//
point										:= 42;
_Camming.camPoints[point].MasterPos			:= 1030.100;
_Camming.camPoints[point].SlavePos			:= 916.716;
_Camming.camPoints[point].PointIndex		:= point;
_Camming.camPoints[point].FunctionType		:= MC_MotionFunctionType.MOTIONFUNCTYPE_POLYNOM5_MM;
_Camming.camPoints[point].PointType			:= MC_MotionPointType.MOTIONPOINTTYPE_MOTION;
_Camming.camPoints[point].RelIndexNextPoint := 1;
_Camming.camPoints[point].SlaveVelo			:= 1.187356;
_Camming.camPoints[point].SlaveAcc			:= 0.01442322;
_Camming.camPoints[point].SlaveJerk			:= 0.00;

//
point										:= 43;
_Camming.camPoints[point].MasterPos			:= 1039.967;
_Camming.camPoints[point].SlavePos			:= 929.194;
_Camming.camPoints[point].PointIndex		:= point;
_Camming.camPoints[point].FunctionType		:= MC_MotionFunctionType.MOTIONFUNCTYPE_POLYNOM5_MM;
_Camming.camPoints[point].PointType			:= MC_MotionPointType.MOTIONPOINTTYPE_MOTION;
_Camming.camPoints[point].RelIndexNextPoint := 1;
_Camming.camPoints[point].SlaveVelo			:= 1.346759;
_Camming.camPoints[point].SlaveAcc			:= 0.01732695;
_Camming.camPoints[point].SlaveJerk			:= 0.00;

//
point										:= 44;
_Camming.camPoints[point].MasterPos			:= 1049.833;
_Camming.camPoints[point].SlavePos			:= 943.327;
_Camming.camPoints[point].PointIndex		:= point;
_Camming.camPoints[point].FunctionType		:= MC_MotionFunctionType.MOTIONFUNCTYPE_POLYNOM5_MM;
_Camming.camPoints[point].PointType			:= MC_MotionPointType.MOTIONPOINTTYPE_MOTION;
_Camming.camPoints[point].RelIndexNextPoint := 1;
_Camming.camPoints[point].SlaveVelo			:= 1.516335;
_Camming.camPoints[point].SlaveAcc			:= 0.01633779;
_Camming.camPoints[point].SlaveJerk			:= 0.00;

//
point										:= 45;
_Camming.camPoints[point].MasterPos			:= 1059.700;
_Camming.camPoints[point].SlavePos			:= 959.017;
_Camming.camPoints[point].PointIndex		:= point;
_Camming.camPoints[point].FunctionType		:= MC_MotionFunctionType.MOTIONFUNCTYPE_POLYNOM5_MM;
_Camming.camPoints[point].PointType			:= MC_MotionPointType.MOTIONPOINTTYPE_MOTION;
_Camming.camPoints[point].RelIndexNextPoint := 1;
_Camming.camPoints[point].SlaveVelo			:= 1.655944;
_Camming.camPoints[point].SlaveAcc			:= 0.01140889;
_Camming.camPoints[point].SlaveJerk			:= 0.00;

//
point										:= 46;
_Camming.camPoints[point].MasterPos			:= 1069.567;
_Camming.camPoints[point].SlavePos			:= 975.802;
_Camming.camPoints[point].PointIndex		:= point;
_Camming.camPoints[point].FunctionType		:= MC_MotionFunctionType.MOTIONFUNCTYPE_POLYNOM5_MM;
_Camming.camPoints[point].PointType			:= MC_MotionPointType.MOTIONPOINTTYPE_MOTION;
_Camming.camPoints[point].RelIndexNextPoint := 1;
_Camming.camPoints[point].SlaveVelo			:= 1.735262;
_Camming.camPoints[point].SlaveAcc			:= 0.00466021;
_Camming.camPoints[point].SlaveJerk			:= 0.00;

//
point										:= 47;
_Camming.camPoints[point].MasterPos			:= 1079.433;
_Camming.camPoints[point].SlavePos			:= 993.059;
_Camming.camPoints[point].PointIndex		:= point;
_Camming.camPoints[point].FunctionType		:= MC_MotionFunctionType.MOTIONFUNCTYPE_POLYNOM5_MM;
_Camming.camPoints[point].PointType			:= MC_MotionPointType.MOTIONPOINTTYPE_MOTION;
_Camming.camPoints[point].RelIndexNextPoint := 1;
_Camming.camPoints[point].SlaveVelo			:= 1.755026;
_Camming.camPoints[point].SlaveAcc			:= 0.00009489;
_Camming.camPoints[point].SlaveJerk			:= 0.00;

//
point										:= 48;
_Camming.camPoints[point].MasterPos			:= 1089.300;
_Camming.camPoints[point].SlavePos			:= 1010.346;
_Camming.camPoints[point].PointIndex		:= point;
_Camming.camPoints[point].FunctionType		:= MC_MotionFunctionType.MOTIONFUNCTYPE_POLYNOM5_MM;
_Camming.camPoints[point].PointType			:= MC_MotionPointType.MOTIONPOINTTYPE_MOTION;
_Camming.camPoints[point].RelIndexNextPoint := 1;
_Camming.camPoints[point].SlaveVelo			:= 1.737154;
_Camming.camPoints[point].SlaveAcc			:= -0.00845956;
_Camming.camPoints[point].SlaveJerk			:= 0.00;

//
point										:= 49;
_Camming.camPoints[point].MasterPos			:= 1099.167;
_Camming.camPoints[point].SlavePos			:= 1026.699;
_Camming.camPoints[point].PointIndex		:= point;
_Camming.camPoints[point].FunctionType		:= MC_MotionFunctionType.MOTIONFUNCTYPE_POLYNOM5_MM;
_Camming.camPoints[point].PointType			:= MC_MotionPointType.MOTIONPOINTTYPE_MOTION;
_Camming.camPoints[point].RelIndexNextPoint := 1;
_Camming.camPoints[point].SlaveVelo			:= 1.547397;
_Camming.camPoints[point].SlaveAcc			:= -0.02615257;
_Camming.camPoints[point].SlaveJerk			:= 0.00;

//
point										:= 50;
_Camming.camPoints[point].MasterPos			:= 1109.033;
_Camming.camPoints[point].SlavePos			:= 1040.717;
_Camming.camPoints[point].PointIndex		:= point;
_Camming.camPoints[point].FunctionType		:= MC_MotionFunctionType.MOTIONFUNCTYPE_POLYNOM5_MM;
_Camming.camPoints[point].PointType			:= MC_MotionPointType.MOTIONPOINTTYPE_MOTION;
_Camming.camPoints[point].RelIndexNextPoint := 1;
_Camming.camPoints[point].SlaveVelo			:= 1.302751;
_Camming.camPoints[point].SlaveAcc			:= -0.02131854;
_Camming.camPoints[point].SlaveJerk			:= 0.00;

//
point										:= 51;
_Camming.camPoints[point].MasterPos			:= 1118.900;
_Camming.camPoints[point].SlavePos			:= 1052.681;
_Camming.camPoints[point].PointIndex		:= point;
_Camming.camPoints[point].FunctionType		:= MC_MotionFunctionType.MOTIONFUNCTYPE_POLYNOM5_MM;
_Camming.camPoints[point].PointType			:= MC_MotionPointType.MOTIONPOINTTYPE_MOTION;
_Camming.camPoints[point].RelIndexNextPoint := 1;
_Camming.camPoints[point].SlaveVelo			:= 1.136789;
_Camming.camPoints[point].SlaveAcc			:= -0.01261846;
_Camming.camPoints[point].SlaveJerk			:= 0.00;

//
point										:= 52;
_Camming.camPoints[point].MasterPos			:= 1128.767;
_Camming.camPoints[point].SlavePos			:= 1063.397;
_Camming.camPoints[point].PointIndex		:= point;
_Camming.camPoints[point].FunctionType		:= MC_MotionFunctionType.MOTIONFUNCTYPE_POLYNOM5_MM;
_Camming.camPoints[point].PointType			:= MC_MotionPointType.MOTIONPOINTTYPE_MOTION;
_Camming.camPoints[point].RelIndexNextPoint := 1;
_Camming.camPoints[point].SlaveVelo			:= 1.045962;
_Camming.camPoints[point].SlaveAcc			:= -0.00622413;
_Camming.camPoints[point].SlaveJerk			:= 0.00;

//
point										:= 53;
_Camming.camPoints[point].MasterPos			:= 1138.633;
_Camming.camPoints[point].SlavePos			:= 1073.492;
_Camming.camPoints[point].PointIndex		:= point;
_Camming.camPoints[point].FunctionType		:= MC_MotionFunctionType.MOTIONFUNCTYPE_POLYNOM5_MM;
_Camming.camPoints[point].PointType			:= MC_MotionPointType.MOTIONPOINTTYPE_MOTION;
_Camming.camPoints[point].RelIndexNextPoint := 1;
_Camming.camPoints[point].SlaveVelo			:= 1.007263;
_Camming.camPoints[point].SlaveAcc			:= -0.00195545;
_Camming.camPoints[point].SlaveJerk			:= 0.00;

//
point										:= 54;
_Camming.camPoints[point].MasterPos			:= 1148.500;
_Camming.camPoints[point].SlavePos			:= 1083.378;
_Camming.camPoints[point].PointIndex		:= point;
_Camming.camPoints[point].FunctionType		:= MC_MotionFunctionType.MOTIONFUNCTYPE_POLYNOM5_MM;
_Camming.camPoints[point].PointType			:= MC_MotionPointType.MOTIONPOINTTYPE_MOTION;
_Camming.camPoints[point].RelIndexNextPoint := 1;
_Camming.camPoints[point].SlaveVelo			:= 1.000000;
_Camming.camPoints[point].SlaveAcc			:= 0.00000000;
_Camming.camPoints[point].SlaveJerk			:= 0.00;

//
point										:= 55;
_Camming.camPoints[point].MasterPos			:= 1416.600;
_Camming.camPoints[point].SlavePos			:= 1351.478;
_Camming.camPoints[point].PointIndex		:= point;
_Camming.camPoints[point].FunctionType		:= MC_MotionFunctionType.MOTIONFUNCTYPE_POLYNOM5_MM;
_Camming.camPoints[point].PointType			:= MC_MotionPointType.MOTIONPOINTTYPE_MOTION;
_Camming.camPoints[point].RelIndexNextPoint := 1;
_Camming.camPoints[point].SlaveVelo			:= 1.000000;
_Camming.camPoints[point].SlaveAcc			:= 0.00000000;
_Camming.camPoints[point].SlaveJerk			:= 0.00;

//
point										:= 56;
_Camming.camPoints[point].MasterPos			:= 1426.495;
_Camming.camPoints[point].SlavePos			:= 1361.354;
_Camming.camPoints[point].PointIndex		:= point;
_Camming.camPoints[point].FunctionType		:= MC_MotionFunctionType.MOTIONFUNCTYPE_POLYNOM5_MM;
_Camming.camPoints[point].PointType			:= MC_MotionPointType.MOTIONPOINTTYPE_MOTION;
_Camming.camPoints[point].RelIndexNextPoint := 1;
_Camming.camPoints[point].SlaveVelo			:= 0.992814;
_Camming.camPoints[point].SlaveAcc			:= -0.00190944;
_Camming.camPoints[point].SlaveJerk			:= 0.00;

//
point										:= 57;
_Camming.camPoints[point].MasterPos			:= 1436.390;
_Camming.camPoints[point].SlavePos			:= 1371.030;
_Camming.camPoints[point].PointIndex		:= point;
_Camming.camPoints[point].FunctionType		:= MC_MotionFunctionType.MOTIONFUNCTYPE_POLYNOM5_MM;
_Camming.camPoints[point].PointType			:= MC_MotionPointType.MOTIONPOINTTYPE_MOTION;
_Camming.camPoints[point].RelIndexNextPoint := 1;
_Camming.camPoints[point].SlaveVelo			:= 0.957206;
_Camming.camPoints[point].SlaveAcc			:= -0.00535633;
_Camming.camPoints[point].SlaveJerk			:= 0.00;

//
point										:= 58;
_Camming.camPoints[point].MasterPos			:= 1446.285;
_Camming.camPoints[point].SlavePos			:= 1380.186;
_Camming.camPoints[point].PointIndex		:= point;
_Camming.camPoints[point].FunctionType		:= MC_MotionFunctionType.MOTIONFUNCTYPE_POLYNOM5_MM;
_Camming.camPoints[point].PointType			:= MC_MotionPointType.MOTIONPOINTTYPE_MOTION;
_Camming.camPoints[point].RelIndexNextPoint := 1;
_Camming.camPoints[point].SlaveVelo			:= 0.888425;
_Camming.camPoints[point].SlaveAcc			:= -0.00834680;
_Camming.camPoints[point].SlaveJerk			:= 0.00;

//
point										:= 59;
_Camming.camPoints[point].MasterPos			:= 1456.180;
_Camming.camPoints[point].SlavePos			:= 1388.538;
_Camming.camPoints[point].PointIndex		:= point;
_Camming.camPoints[point].FunctionType		:= MC_MotionFunctionType.MOTIONFUNCTYPE_POLYNOM5_MM;
_Camming.camPoints[point].PointType			:= MC_MotionPointType.MOTIONPOINTTYPE_MOTION;
_Camming.camPoints[point].RelIndexNextPoint := 1;
_Camming.camPoints[point].SlaveVelo			:= 0.797621;
_Camming.camPoints[point].SlaveAcc			:= -0.00966634;
_Camming.camPoints[point].SlaveJerk			:= 0.00;

//
point										:= 60;
_Camming.camPoints[point].MasterPos			:= 1466.075;
_Camming.camPoints[point].SlavePos			:= 1395.962;
_Camming.camPoints[point].PointIndex		:= point;
_Camming.camPoints[point].FunctionType		:= MC_MotionFunctionType.MOTIONFUNCTYPE_POLYNOM5_MM;
_Camming.camPoints[point].PointType			:= MC_MotionPointType.MOTIONPOINTTYPE_MOTION;
_Camming.camPoints[point].RelIndexNextPoint := 1;
_Camming.camPoints[point].SlaveVelo			:= 0.704244;
_Camming.camPoints[point].SlaveAcc			:= -0.00885381;
_Camming.camPoints[point].SlaveJerk			:= 0.00;

//
point										:= 61;
_Camming.camPoints[point].MasterPos			:= 1475.970;
_Camming.camPoints[point].SlavePos			:= 1402.534;
_Camming.camPoints[point].PointIndex		:= point;
_Camming.camPoints[point].FunctionType		:= MC_MotionFunctionType.MOTIONFUNCTYPE_POLYNOM5_MM;
_Camming.camPoints[point].PointType			:= MC_MotionPointType.MOTIONPOINTTYPE_MOTION;
_Camming.camPoints[point].RelIndexNextPoint := 1;
_Camming.camPoints[point].SlaveVelo			:= 0.628520;
_Camming.camPoints[point].SlaveAcc			:= -0.00621225;
_Camming.camPoints[point].SlaveJerk			:= 0.00;

//
point										:= 62;
_Camming.camPoints[point].MasterPos			:= 1485.865;
_Camming.camPoints[point].SlavePos			:= 1408.505;
_Camming.camPoints[point].PointIndex		:= point;
_Camming.camPoints[point].FunctionType		:= MC_MotionFunctionType.MOTIONFUNCTYPE_POLYNOM5_MM;
_Camming.camPoints[point].PointType			:= MC_MotionPointType.MOTIONPOINTTYPE_MOTION;
_Camming.camPoints[point].RelIndexNextPoint := 1;
_Camming.camPoints[point].SlaveVelo			:= 0.583944;
_Camming.camPoints[point].SlaveAcc			:= -0.00279152;
_Camming.camPoints[point].SlaveJerk			:= 0.00;

//
point										:= 63;
_Camming.camPoints[point].MasterPos			:= 1495.760;
_Camming.camPoints[point].SlavePos			:= 1414.195;
_Camming.camPoints[point].PointIndex		:= point;
_Camming.camPoints[point].FunctionType		:= MC_MotionFunctionType.MOTIONFUNCTYPE_POLYNOM5_MM;
_Camming.camPoints[point].PointType			:= MC_MotionPointType.MOTIONPOINTTYPE_MOTION;
_Camming.camPoints[point].RelIndexNextPoint := 1;
_Camming.camPoints[point].SlaveVelo			:= 0.570311;
_Camming.camPoints[point].SlaveAcc			:= -0.00028497;
_Camming.camPoints[point].SlaveJerk			:= 0.00;

//
point										:= 64;
_Camming.camPoints[point].MasterPos			:= 1505.655;
_Camming.camPoints[point].SlavePos			:= 1419.834;
_Camming.camPoints[point].PointIndex		:= point;
_Camming.camPoints[point].FunctionType		:= MC_MotionFunctionType.MOTIONFUNCTYPE_POLYNOM5_MM;
_Camming.camPoints[point].PointType			:= MC_MotionPointType.MOTIONPOINTTYPE_MOTION;
_Camming.camPoints[point].RelIndexNextPoint := 1;
_Camming.camPoints[point].SlaveVelo			:= 0.569785;
_Camming.camPoints[point].SlaveAcc			:= -0.00000641;
_Camming.camPoints[point].SlaveJerk			:= 0.00;

//
point										:= 65;
_Camming.camPoints[point].MasterPos			:= 1515.550;
_Camming.camPoints[point].SlavePos			:= 1425.476;
_Camming.camPoints[point].PointIndex		:= point;
_Camming.camPoints[point].FunctionType		:= MC_MotionFunctionType.MOTIONFUNCTYPE_POLYNOM5_MM;
_Camming.camPoints[point].PointType			:= MC_MotionPointType.MOTIONPOINTTYPE_MOTION;
_Camming.camPoints[point].RelIndexNextPoint := 1;
_Camming.camPoints[point].SlaveVelo			:= 0.571122;
_Camming.camPoints[point].SlaveAcc			:= 0.00033576;
_Camming.camPoints[point].SlaveJerk			:= 0.00;

//
point										:= 66;
_Camming.camPoints[point].MasterPos			:= 1525.445;
_Camming.camPoints[point].SlavePos			:= 1431.153;
_Camming.camPoints[point].PointIndex		:= point;
_Camming.camPoints[point].FunctionType		:= MC_MotionFunctionType.MOTIONFUNCTYPE_POLYNOM5_MM;
_Camming.camPoints[point].PointType			:= MC_MotionPointType.MOTIONPOINTTYPE_MOTION;
_Camming.camPoints[point].RelIndexNextPoint := 1;
_Camming.camPoints[point].SlaveVelo			:= 0.577454;
_Camming.camPoints[point].SlaveAcc			:= 0.00098723;
_Camming.camPoints[point].SlaveJerk			:= 0.00;

//
point										:= 67;
_Camming.camPoints[point].MasterPos			:= 1535.340;
_Camming.camPoints[point].SlavePos			:= 1436.929;
_Camming.camPoints[point].PointIndex		:= point;
_Camming.camPoints[point].FunctionType		:= MC_MotionFunctionType.MOTIONFUNCTYPE_POLYNOM5_MM;
_Camming.camPoints[point].PointType			:= MC_MotionPointType.MOTIONPOINTTYPE_MOTION;
_Camming.camPoints[point].RelIndexNextPoint := 1;
_Camming.camPoints[point].SlaveVelo			:= 0.591500;
_Camming.camPoints[point].SlaveAcc			:= 0.00188997;
_Camming.camPoints[point].SlaveJerk			:= 0.00;

//
point										:= 68;
_Camming.camPoints[point].MasterPos			:= 1545.235;
_Camming.camPoints[point].SlavePos			:= 1442.892;
_Camming.camPoints[point].PointIndex		:= point;
_Camming.camPoints[point].FunctionType		:= MC_MotionFunctionType.MOTIONFUNCTYPE_POLYNOM5_MM;
_Camming.camPoints[point].PointType			:= MC_MotionPointType.MOTIONPOINTTYPE_MOTION;
_Camming.camPoints[point].RelIndexNextPoint := 1;
_Camming.camPoints[point].SlaveVelo			:= 0.615664;
_Camming.camPoints[point].SlaveAcc			:= 0.00303751;
_Camming.camPoints[point].SlaveJerk			:= 0.00;

//
point										:= 69;
_Camming.camPoints[point].MasterPos			:= 1555.130;
_Camming.camPoints[point].SlavePos			:= 1449.155;
_Camming.camPoints[point].PointIndex		:= point;
_Camming.camPoints[point].FunctionType		:= MC_MotionFunctionType.MOTIONFUNCTYPE_POLYNOM5_MM;
_Camming.camPoints[point].PointType			:= MC_MotionPointType.MOTIONPOINTTYPE_MOTION;
_Camming.camPoints[point].RelIndexNextPoint := 1;
_Camming.camPoints[point].SlaveVelo			:= 0.652442;
_Camming.camPoints[point].SlaveAcc			:= 0.00443439;
_Camming.camPoints[point].SlaveJerk			:= 0.00;

//
point										:= 70;
_Camming.camPoints[point].MasterPos			:= 1565.025;
_Camming.camPoints[point].SlavePos			:= 1455.854;
_Camming.camPoints[point].PointIndex		:= point;
_Camming.camPoints[point].FunctionType		:= MC_MotionFunctionType.MOTIONFUNCTYPE_POLYNOM5_MM;
_Camming.camPoints[point].PointType			:= MC_MotionPointType.MOTIONPOINTTYPE_MOTION;
_Camming.camPoints[point].RelIndexNextPoint := 1;
_Camming.camPoints[point].SlaveVelo			:= 0.704402;
_Camming.camPoints[point].SlaveAcc			:= 0.00609093;
_Camming.camPoints[point].SlaveJerk			:= 0.00;

//
point										:= 71;
_Camming.camPoints[point].MasterPos			:= 1574.920;
_Camming.camPoints[point].SlavePos			:= 1463.150;
_Camming.camPoints[point].PointIndex		:= point;
_Camming.camPoints[point].FunctionType		:= MC_MotionFunctionType.MOTIONFUNCTYPE_POLYNOM5_MM;
_Camming.camPoints[point].PointType			:= MC_MotionPointType.MOTIONPOINTTYPE_MOTION;
_Camming.camPoints[point].RelIndexNextPoint := 1;
_Camming.camPoints[point].SlaveVelo			:= 0.773096;
_Camming.camPoints[point].SlaveAcc			:= 0.00774577;
_Camming.camPoints[point].SlaveJerk			:= 0.00;

//
point										:= 72;
_Camming.camPoints[point].MasterPos			:= 1584.815;
_Camming.camPoints[point].SlavePos			:= 1471.200;
_Camming.camPoints[point].PointIndex		:= point;
_Camming.camPoints[point].FunctionType		:= MC_MotionFunctionType.MOTIONFUNCTYPE_POLYNOM5_MM;
_Camming.camPoints[point].PointType			:= MC_MotionPointType.MOTIONPOINTTYPE_MOTION;
_Camming.camPoints[point].RelIndexNextPoint := 1;
_Camming.camPoints[point].SlaveVelo			:= 0.855433;
_Camming.camPoints[point].SlaveAcc			:= 0.00865192;
_Camming.camPoints[point].SlaveJerk			:= 0.00;

//
point										:= 73;
_Camming.camPoints[point].MasterPos			:= 1594.710;
_Camming.camPoints[point].SlavePos			:= 1480.077;
_Camming.camPoints[point].PointIndex		:= point;
_Camming.camPoints[point].FunctionType		:= MC_MotionFunctionType.MOTIONFUNCTYPE_POLYNOM5_MM;
_Camming.camPoints[point].PointType			:= MC_MotionPointType.MOTIONPOINTTYPE_MOTION;
_Camming.camPoints[point].RelIndexNextPoint := 1;
_Camming.camPoints[point].SlaveVelo			:= 0.936508;
_Camming.camPoints[point].SlaveAcc			:= 0.00721864;
_Camming.camPoints[point].SlaveJerk			:= 0.00;

//
point										:= 74;
_Camming.camPoints[point].MasterPos			:= 1604.605;
_Camming.camPoints[point].SlavePos			:= 1489.636;
_Camming.camPoints[point].PointIndex		:= point;
_Camming.camPoints[point].FunctionType		:= MC_MotionFunctionType.MOTIONFUNCTYPE_POLYNOM5_MM;
_Camming.camPoints[point].PointType			:= MC_MotionPointType.MOTIONPOINTTYPE_MOTION;
_Camming.camPoints[point].RelIndexNextPoint := 1;
_Camming.camPoints[point].SlaveVelo			:= 0.988558;
_Camming.camPoints[point].SlaveAcc			:= 0.00301892;
_Camming.camPoints[point].SlaveJerk			:= 0.00;

//
point										:= 75;
_Camming.camPoints[point].MasterPos			:= 1614.500;
_Camming.camPoints[point].SlavePos			:= 1499.500;
_Camming.camPoints[point].PointIndex		:= point;
_Camming.camPoints[point].FunctionType		:= MC_MotionFunctionType.MOTIONFUNCTYPE_POLYNOM5_MM;
_Camming.camPoints[point].PointType			:= MC_MotionPointType.MOTIONPOINTTYPE_MOTION;
_Camming.camPoints[point].RelIndexNextPoint := 1;
_Camming.camPoints[point].SlaveVelo			:= 1.000000;
_Camming.camPoints[point].SlaveAcc			:= 0.00000000;
_Camming.camPoints[point].SlaveJerk			:= 0.00;

//
point										:= 76;
_Camming.camPoints[point].MasterPos			:= 1680.000;
_Camming.camPoints[point].SlavePos			:= 1565.000;
_Camming.camPoints[point].PointIndex		:= point;
_Camming.camPoints[point].FunctionType		:= MC_MotionFunctionType.MOTIONFUNCTYPE_POLYNOM5_MM;
_Camming.camPoints[point].PointType			:= MC_MotionPointType.MOTIONPOINTTYPE_MOTION;
_Camming.camPoints[point].RelIndexNextPoint := 0;
_Camming.camPoints[point].SlaveVelo			:= 1.000000;
_Camming.camPoints[point].SlaveAcc			:= 0.00000000;
_Camming.camPoints[point].SlaveJerk			:= 0.00;
END_METHOD

METHOD Old
VAR_INPUT
END_VAR
IF NOT _Custom THEN
	point										:= 1;
	_Camming.camPoints[point].MasterPos			:= 250;
	_Camming.camPoints[point].SlavePos			:= 135;
	_Camming.camPoints[point].PointIndex		:= point;
	_Camming.camPoints[point].FunctionType		:= MC_MotionFunctionType.MOTIONFUNCTYPE_POLYNOM1;
	_Camming.camPoints[point].PointType			:= MC_MotionPointType.MOTIONPOINTTYPE_ACTIVATION;
	_Camming.camPoints[point].RelIndexNextPoint := 1;
	_Camming.camPoints[point].SlaveVelo			:= 0.00;
	_Camming.camPoints[point].SlaveAcc			:= 0.00;
	_Camming.camPoints[point].SlaveJerk			:= 0.00;

	//
	point										:= 2;
	_Camming.camPoints[point].MasterPos			:= 291;
	_Camming.camPoints[point].SlavePos			:= 176;
	_Camming.camPoints[point].PointIndex		:= point;
	_Camming.camPoints[point].FunctionType		:= MC_MotionFunctionType.MOTIONFUNCTYPE_POLYNOM5_MM;
	_Camming.camPoints[point].PointType			:= MC_MotionPointType.MOTIONPOINTTYPE_ACTIVATION;
	_Camming.camPoints[point].RelIndexNextPoint := 1;
	_Camming.camPoints[point].SlaveVelo			:= 0.00;
	_Camming.camPoints[point].SlaveAcc			:= 0.00;
	_Camming.camPoints[point].SlaveJerk			:= 0.00;

	//
	point										:= 3;
	_Camming.camPoints[point].MasterPos			:= 377.1;
	_Camming.camPoints[point].SlavePos			:= 317.3;
	_Camming.camPoints[point].PointIndex		:= point;
	_Camming.camPoints[point].FunctionType		:= MC_MotionFunctionType.MOTIONFUNCTYPE_POLYNOM1;
	_Camming.camPoints[point].PointType			:= MC_MotionPointType.MOTIONPOINTTYPE_ACTIVATION;
	_Camming.camPoints[point].RelIndexNextPoint := 1;
	_Camming.camPoints[point].SlaveVelo			:= 0.00;
	_Camming.camPoints[point].SlaveAcc			:= 0.00;
	_Camming.camPoints[point].SlaveJerk			:= 0.00;

	//
	point										:= 4;
	_Camming.camPoints[point].MasterPos			:= 704.5;
	_Camming.camPoints[point].SlavePos			:= 643.0;
	_Camming.camPoints[point].PointIndex		:= point;
	_Camming.camPoints[point].FunctionType		:= MC_MotionFunctionType.MOTIONFUNCTYPE_POLYNOM5_MM;
	_Camming.camPoints[point].PointType			:= MC_MotionPointType.MOTIONPOINTTYPE_ACTIVATION;
	_Camming.camPoints[point].RelIndexNextPoint := 1;
	_Camming.camPoints[point].SlaveVelo			:= 0.00;
	_Camming.camPoints[point].SlaveAcc			:= 0.00;
	_Camming.camPoints[point].SlaveJerk			:= 0.00;

	//
	point										:= 5;
	_Camming.camPoints[point].MasterPos			:= 815;
	_Camming.camPoints[point].SlavePos			:= 700;
	_Camming.camPoints[point].PointIndex		:= point;
	_Camming.camPoints[point].FunctionType		:= MC_MotionFunctionType.MOTIONFUNCTYPE_POLYNOM1;
	_Camming.camPoints[point].PointType			:= MC_MotionPointType.MOTIONPOINTTYPE_ACTIVATION;
	_Camming.camPoints[point].RelIndexNextPoint := 1;
	_Camming.camPoints[point].SlaveVelo			:= 0.00;
	_Camming.camPoints[point].SlaveAcc			:= 0.00;
	_Camming.camPoints[point].SlaveJerk			:= 0.00;

	//
	point										:= 6;
	_Camming.camPoints[point].MasterPos			:= 1037;
	_Camming.camPoints[point].SlavePos			:= 922;
	_Camming.camPoints[point].PointIndex		:= point;
	_Camming.camPoints[point].FunctionType		:= MC_MotionFunctionType.MOTIONFUNCTYPE_POLYNOM5_MM;
	_Camming.camPoints[point].PointType			:= MC_MotionPointType.MOTIONPOINTTYPE_ACTIVATION;
	_Camming.camPoints[point].RelIndexNextPoint := 1;
	_Camming.camPoints[point].SlaveVelo			:= 0.00;
	_Camming.camPoints[point].SlaveAcc			:= 0.00;
	_Camming.camPoints[point].SlaveJerk			:= 0.00;

	//
	point										:= 7;
	_Camming.camPoints[point].MasterPos			:= 1117;
	_Camming.camPoints[point].SlavePos			:= 1057;
	_Camming.camPoints[point].PointIndex		:= point;
	_Camming.camPoints[point].FunctionType		:= MC_MotionFunctionType.MOTIONFUNCTYPE_POLYNOM1;
	_Camming.camPoints[point].PointType			:= MC_MotionPointType.MOTIONPOINTTYPE_ACTIVATION;
	_Camming.camPoints[point].RelIndexNextPoint := 1;
	_Camming.camPoints[point].SlaveVelo			:= 0.00;
	_Camming.camPoints[point].SlaveAcc			:= 0.00;
	_Camming.camPoints[point].SlaveJerk			:= 0.00;

	//
	point										:= 8;
	_Camming.camPoints[point].MasterPos			:= 1449;
	_Camming.camPoints[point].SlavePos			:= 1389;
	_Camming.camPoints[point].PointIndex		:= point;
	_Camming.camPoints[point].FunctionType		:= MC_MotionFunctionType.MOTIONFUNCTYPE_POLYNOM5_MM;
	_Camming.camPoints[point].PointType			:= MC_MotionPointType.MOTIONPOINTTYPE_ACTIVATION;
	_Camming.camPoints[point].RelIndexNextPoint := 1;
	_Camming.camPoints[point].SlaveVelo			:= 0.00;
	_Camming.camPoints[point].SlaveAcc			:= 0.00;
	_Camming.camPoints[point].SlaveJerk			:= 0.00;

	//
	point										:= 9;
	_Camming.camPoints[point].MasterPos			:= 1589;
	_Camming.camPoints[point].SlavePos			:= 1474;
	_Camming.camPoints[point].PointIndex		:= point;
	_Camming.camPoints[point].FunctionType		:= MC_MotionFunctionType.MOTIONFUNCTYPE_POLYNOM1;
	_Camming.camPoints[point].PointType			:= MC_MotionPointType.MOTIONPOINTTYPE_ACTIVATION;
	_Camming.camPoints[point].RelIndexNextPoint := 1;
	_Camming.camPoints[point].SlaveVelo			:= 0.00;
	_Camming.camPoints[point].SlaveAcc			:= 0.00;
	_Camming.camPoints[point].SlaveJerk			:= 0.00;

	//
	point										:= 10;
	_Camming.camPoints[point].MasterPos			:= 1750;
	_Camming.camPoints[point].SlavePos			:= 1635;
	_Camming.camPoints[point].PointIndex		:= point;
	_Camming.camPoints[point].FunctionType		:= MC_MotionFunctionType.MOTIONFUNCTYPE_POLYNOM1;
	_Camming.camPoints[point].PointType			:= MC_MotionPointType.MOTIONPOINTTYPE_ACTIVATION;
	_Camming.camPoints[point].RelIndexNextPoint := 0;
	_Camming.camPoints[point].SlaveVelo			:= 0.00;
	_Camming.camPoints[point].SlaveAcc			:= 0.00;
	_Camming.camPoints[point].SlaveJerk			:= 0.00;
END_IF
END_METHOD

METHOD Reset
SetStep(_State, 0);
_Camming.camTableSelect(CamTable := _Camming.camRef, Execute := FALSE);
END_METHOD

METHOD Start
NextStep(_State);
END_METHOD

{warning 'Add method implementation '}
METHOD Stop
END_METHOD

END_FUNCTION_BLOCK

// ---- Tests/CamCurveCompTest/CamCurveComp.TcPOU
FUNCTION_BLOCK CamCurveComp IMPLEMENTS I_CamBuildSequence
VAR
	_State			: UDINT;
	_Front			: I_XtsMover;
	_Rear			: I_XtsMover;
	_Virtual		: I_XtsMover;
	_StartPosition	: LREAL := 194;
	_Speed			: LREAL := 200;
	_Acc			: LREAL := 10_000;
	_Dec			: LREAL := 10_000;
	_Jerk			: LREAL := 100_000;
	_Camming		: ST_Camming;
	_Scaling		: ST_CamScalingData;
	_Offset			: DINT;
	_NumOfRotations : LREAL := 1;
END_VAR

{attribute 'monitoring' := 'call'}
{warning 'Add property implementation'}
PROPERTY Busy : BOOL
GET
END_GET
END_PROPERTY

METHOD CyclicLogic
CASE _State OF
	0:
	10:
		_Virtual.MoveToPosition(Position := _StartPosition);
		NextMinorStep(_State);

	11:
		IF NOT _Virtual.CurrentTask.Busy AND NOT _Virtual.CurrentTask.Error THEN
			NextStep(_State);
		END_IF

	20:
		_Camming.camIn(Master	  := _Front.Axis,
					   Slave	  := _Rear.Axis,
					   Execute	  := TRUE,
					   CamTableID := 1);

		IF NOT _Camming.camIn.Busy AND NOT _Camming.camIn.Error THEN
			_Camming.camIn(Master := _Front.Axis, Slave := _Rear.Axis, Execute := FALSE);
			NextStep(_State);
		END_IF

	31:
		_Virtual.Parameters.Velocity	 := _Speed;
		_Virtual.Parameters.Acceleration := _Acc;
		_Virtual.Parameters.Deceleration := _Dec;
		_Virtual.Parameters.Jerk		 := _Jerk;
		_Virtual.MoveRelative(1500 * _NumOfRotations);
		NextMinorStep(_State);

	32:
		IF NOT _Virtual.CurrentTask.Busy AND NOT _Virtual.CurrentTask.Error THEN
			NextStep(_State);
		END_IF

	40:
		_Camming.camOut(Slave := _Rear.Axis, Execute := TRUE);
		IF NOT _Camming.camOut.Busy AND NOT _Camming.camOut.Error THEN
			_Camming.camOut(Slave := _Rear.Axis, Execute := FALSE);
			SetStep(_State, 0);
		END_IF
END_CASE
END_METHOD

PROPERTY FrontMover : I_XtsMover
GET
FrontMover := _Front;
END_GET
SET
_Front := FrontMover;
END_SET
END_PROPERTY

PROPERTY RearMover : I_XtsMover
GET
RearMover := _Rear;
END_GET
SET
_Rear := RearMover;
END_SET
END_PROPERTY

METHOD Reset
_Camming.camIn(Master := _Front.Axis, Slave := _Rear.Axis, Execute := FALSE);
_Virtual.Reset();
SetStep(_State, 0);
END_METHOD

METHOD Start
NextStep(_State);
END_METHOD

{warning 'Add method implementation '}
METHOD Stop
END_METHOD

PROPERTY VirtualMover : I_XtsMover
GET
VirtualMover := _Virtual;
END_GET
SET
_Virtual := VirtualMover;
END_SET
END_PROPERTY

END_FUNCTION_BLOCK

// ---- Tests/CamBuild/SplitCamBuild.TcPOU
FUNCTION_BLOCK SplitCamBuild IMPLEMENTS I_CamBuildSequence
VAR
	_State	 : UDINT;
	_Camming : ST_Camming;
	point	 : UDINT;
	_Custom	 : BOOL;
END_VAR

{attribute 'monitoring' := 'call'}
PROPERTY Busy : BOOL
GET
Busy := _State <> 0;
END_GET
END_PROPERTY

METHOD CyclicLogic
VAR_INPUT
END_VAR
CASE _State OF
	0:
	10:
		point										:= 1;
		_Camming.camPoints[point].MasterPos			:= 0;
		_Camming.camPoints[point].SlavePos			:= 0;
		_Camming.camPoints[point].PointIndex		:= point;
		_Camming.camPoints[point].FunctionType		:= MC_MotionFunctionType.MOTIONFUNCTYPE_POLYNOM1;
		_Camming.camPoints[point].PointType			:= MC_MotionPointType.MOTIONPOINTTYPE_ACTIVATION;
		_Camming.camPoints[point].RelIndexNextPoint := 1;
		_Camming.camPoints[point].SlaveVelo			:= 0.00;
		_Camming.camPoints[point].SlaveAcc			:= 0.00;
		_Camming.camPoints[point].SlaveJerk			:= 0.00;

		//
		point										:= 2;
		_Camming.camPoints[point].MasterPos			:= 1;
		_Camming.camPoints[point].SlavePos			:= 1;
		_Camming.camPoints[point].PointIndex		:= point;
		_Camming.camPoints[point].FunctionType		:= MC_MotionFunctionType.MOTIONFUNCTYPE_POLYNOM1;
		_Camming.camPoints[point].PointType			:= MC_MotionPointType.MOTIONPOINTTYPE_MOTION;
		_Camming.camPoints[point].RelIndexNextPoint := 0;
		_Camming.camPoints[point].SlaveVelo			:= 0.00;
		_Camming.camPoints[point].SlaveAcc			:= 0.00;
		_Camming.camPoints[point].SlaveJerk			:= 0.00;

		//
		_Camming.camRef.NoOfColumns := 1;
		_Camming.camRef.NoOfRows	:= point;
		_Camming.camRef.TableType	:= MC_TableType.MC_TABLETYPE_MOTIONFUNCTION;
		_Camming.camRef.ArraySize	:= SIZEOF(_Camming.camPoints);
		_Camming.camRef.pArray		:= ADR(_Camming.camPoints);

		//
		_Camming.camTableSelect(CamTable   := _Camming.camRef,
								Execute	   := TRUE,
								Periodic   := TRUE,
								CamTableID := 1);

		IF _Camming.camTableSelect.Done THEN
			Trace.Info(__POUNAME(), 'Curve Cam Built - ID 1');
			_Camming.camTableSelect(CamTable := _Camming.camRef, Execute := FALSE);
			MEMSET(ADR(_Camming.camPoints), 0, SIZEOF(_Camming.camPoints));
			NextStep(_State);
		END_IF

	20:
		point										:= 1;
		_Camming.camPoints[point].MasterPos			:= 250;
		_Camming.camPoints[point].SlavePos			:= 135;
		_Camming.camPoints[point].PointIndex		:= point;
		_Camming.camPoints[point].FunctionType		:= MC_MotionFunctionType.MOTIONFUNCTYPE_POLYNOM1;
		_Camming.camPoints[point].PointType			:= MC_MotionPointType.MOTIONPOINTTYPE_ACTIVATION;
		_Camming.camPoints[point].RelIndexNextPoint := 1;
		_Camming.camPoints[point].SlaveVelo			:= 0.00;
		_Camming.camPoints[point].SlaveAcc			:= 0.00;
		_Camming.camPoints[point].SlaveJerk			:= 0.00;

		//
		point										:= 2;
		_Camming.camPoints[point].MasterPos			:= 281;
		_Camming.camPoints[point].SlavePos			:= 169;
		_Camming.camPoints[point].PointIndex		:= point;
		_Camming.camPoints[point].FunctionType		:= MC_MotionFunctionType.MOTIONFUNCTYPE_POLYNOM5_MM;
		_Camming.camPoints[point].PointType			:= MC_MotionPointType.MOTIONPOINTTYPE_MOTION;
		_Camming.camPoints[point].RelIndexNextPoint := 1;
		_Camming.camPoints[point].SlaveVelo			:= 0.00;
		_Camming.camPoints[point].SlaveAcc			:= 0.00;
		_Camming.camPoints[point].SlaveJerk			:= 0.00;

		//
		point										:= 3;
		_Camming.camPoints[point].MasterPos			:= 329.4;
		_Camming.camPoints[point].SlavePos			:= 242.7;
		_Camming.camPoints[point].PointIndex		:= point;
		_Camming.camPoints[point].FunctionType		:= MC_MotionFunctionType.MOTIONFUNCTYPE_POLYNOM1;
		_Camming.camPoints[point].PointType			:= MC_MotionPointType.MOTIONPOINTTYPE_MOTION;
		_Camming.camPoints[point].RelIndexNextPoint := 1;
		_Camming.camPoints[point].SlaveVelo			:= 0.00;
		_Camming.camPoints[point].SlaveAcc			:= 0.00;
		_Camming.camPoints[point].SlaveJerk			:= 0.00;

		//
		point										:= 4;
		_Camming.camPoints[point].MasterPos			:= 353.6;
		_Camming.camPoints[point].SlavePos			:= 288.8;
		_Camming.camPoints[point].PointIndex		:= point;
		_Camming.camPoints[point].FunctionType		:= MC_MotionFunctionType.MOTIONFUNCTYPE_POLYNOM5_MM;
		_Camming.camPoints[point].PointType			:= MC_MotionPointType.MOTIONPOINTTYPE_MOTION;
		_Camming.camPoints[point].RelIndexNextPoint := 1;
		_Camming.camPoints[point].SlaveVelo			:= 0.00;
		_Camming.camPoints[point].SlaveAcc			:= 0.00;
		_Camming.camPoints[point].SlaveJerk			:= 0.00;

		//
		point										:= 5;
		_Camming.camPoints[point].MasterPos			:= 412;
		_Camming.camPoints[point].SlavePos			:= 349.6;
		_Camming.camPoints[point].PointIndex		:= point;
		_Camming.camPoints[point].FunctionType		:= MC_MotionFunctionType.MOTIONFUNCTYPE_POLYNOM1;
		_Camming.camPoints[point].PointType			:= MC_MotionPointType.MOTIONPOINTTYPE_MOTION;
		_Camming.camPoints[point].RelIndexNextPoint := 1;
		_Camming.camPoints[point].SlaveVelo			:= 0.00;
		_Camming.camPoints[point].SlaveAcc			:= 0.00;
		_Camming.camPoints[point].SlaveJerk			:= 0.00;

		//
		point										:= 6;
		_Camming.camPoints[point].MasterPos			:= 700;
		_Camming.camPoints[point].SlavePos			:= 641;
		_Camming.camPoints[point].PointIndex		:= point;
		_Camming.camPoints[point].FunctionType		:= MC_MotionFunctionType.MOTIONFUNCTYPE_POLYNOM5_MM;
		_Camming.camPoints[point].PointType			:= MC_MotionPointType.MOTIONPOINTTYPE_MOTION;
		_Camming.camPoints[point].RelIndexNextPoint := 1;
		_Camming.camPoints[point].SlaveVelo			:= 0.00;
		_Camming.camPoints[point].SlaveAcc			:= 0.00;
		_Camming.camPoints[point].SlaveJerk			:= 0.00;

		//
		point										:= 7;
		_Camming.camPoints[point].MasterPos			:= 727.3;
		_Camming.camPoints[point].SlavePos			:= 657.6;
		_Camming.camPoints[point].PointIndex		:= point;
		_Camming.camPoints[point].FunctionType		:= MC_MotionFunctionType.MOTIONFUNCTYPE_POLYNOM1;
		_Camming.camPoints[point].PointType			:= MC_MotionPointType.MOTIONPOINTTYPE_MOTION;
		_Camming.camPoints[point].RelIndexNextPoint := 1;
		_Camming.camPoints[point].SlaveVelo			:= 0.00;
		_Camming.camPoints[point].SlaveAcc			:= 0.00;
		_Camming.camPoints[point].SlaveJerk			:= 0.00;

		//
		point										:= 8;
		_Camming.camPoints[point].MasterPos			:= 791.4;
		_Camming.camPoints[point].SlavePos			:= 690.2;
		_Camming.camPoints[point].PointIndex		:= point;
		_Camming.camPoints[point].FunctionType		:= MC_MotionFunctionType.MOTIONFUNCTYPE_POLYNOM5_MM;
		_Camming.camPoints[point].PointType			:= MC_MotionPointType.MOTIONPOINTTYPE_MOTION;
		_Camming.camPoints[point].RelIndexNextPoint := 1;
		_Camming.camPoints[point].SlaveVelo			:= 0.00;
		_Camming.camPoints[point].SlaveAcc			:= 0.00;
		_Camming.camPoints[point].SlaveJerk			:= 0.00;

		//
		point										:= 9;
		_Camming.camPoints[point].MasterPos			:= 834;
		_Camming.camPoints[point].SlavePos			:= 723;
		_Camming.camPoints[point].PointIndex		:= point;
		_Camming.camPoints[point].FunctionType		:= MC_MotionFunctionType.MOTIONFUNCTYPE_POLYNOM1;
		_Camming.camPoints[point].PointType			:= MC_MotionPointType.MOTIONPOINTTYPE_MOTION;
		_Camming.camPoints[point].RelIndexNextPoint := 1;
		_Camming.camPoints[point].SlaveVelo			:= 0.00;
		_Camming.camPoints[point].SlaveAcc			:= 0.00;
		_Camming.camPoints[point].SlaveJerk			:= 0.00;

		//
		point										:= 10;
		_Camming.camPoints[point].MasterPos			:= 865;
		_Camming.camPoints[point].SlavePos			:= 750;
		_Camming.camPoints[point].PointIndex		:= point;
		_Camming.camPoints[point].FunctionType		:= MC_MotionFunctionType.MOTIONFUNCTYPE_POLYNOM5_MM;
		_Camming.camPoints[point].PointType			:= MC_MotionPointType.MOTIONPOINTTYPE_MOTION;
		_Camming.camPoints[point].RelIndexNextPoint := 0;
		_Camming.camPoints[point].SlaveVelo			:= 0.00;
		_Camming.camPoints[point].SlaveAcc			:= 0.00;
		_Camming.camPoints[point].SlaveJerk			:= 0.00;

		//
		_Camming.camRef.NoOfColumns := 1;
		_Camming.camRef.NoOfRows	:= point;
		_Camming.camRef.TableType	:= MC_TableType.MC_TABLETYPE_MOTIONFUNCTION;
		_Camming.camRef.ArraySize	:= SIZEOF(_Camming.camPoints);
		_Camming.camRef.pArray		:= ADR(_Camming.camPoints);

		//
		_Camming.camTableSelect(CamTable   := _Camming.camRef,
								Execute	   := TRUE,
								Periodic   := FALSE,
								CamTableID := 2);

		IF _Camming.camTableSelect.Done THEN
			Trace.Info(__POUNAME(), 'Curve Cam Built - ID 2');
			_Camming.camTableSelect(CamTable := _Camming.camRef, Execute := FALSE);
			SetStep(_State, 0);
		END_IF
END_CASE
END_METHOD

METHOD Reset
SetStep(_State, 0);
_Camming.camTableSelect(CamTable := _Camming.camRef, Execute := FALSE);
END_METHOD

METHOD Start
NextStep(_State);
END_METHOD

{warning 'Add method implementation '}
METHOD Stop
END_METHOD

END_FUNCTION_BLOCK

// ---- Tests/CamCurveCompTest/SplitCamRun.TcPOU
FUNCTION_BLOCK SplitCamRun IMPLEMENTS I_CamBuildSequence
VAR
	_State			: UDINT;
	_Front			: I_XtsMover;
	_Rear			: I_XtsMover;
	_Virtual		: I_XtsMover;
	_StartPosition	: LREAL := 59;
	_Speed			: LREAL := 200;
	_Acc			: LREAL := 10_000;
	_Dec			: LREAL := 10_000;
	_Jerk			: LREAL := 100_000;
	_Camming		: ST_Camming;
	_Scaling		: ST_CamScalingData;
	_Offset			: DINT;
	_Distance		: LREAL := 100;
	_NumOfRotations : LREAL := 1;
END_VAR

{attribute 'monitoring' := 'call'}
{warning 'Add property implementation'}
PROPERTY Busy : BOOL
GET
END_GET
END_PROPERTY

METHOD CyclicLogic
CASE _State OF
	0:
	10:
		_Virtual.MoveToPosition(Position := _StartPosition, Direction := _Virtual.Parameters.Direction);
		NextMinorStep(_State);

	11:
		IF NOT _Virtual.CurrentTask.Busy AND NOT _Virtual.CurrentTask.Error THEN
			NextStep(_State);
		END_IF

	20:
		//_Camming.camIn.Options.CamOperationMode := CAMOPERATIONMODE_DEFAULT;
		_Camming.camIn.ActivationPosition		:= 0;
		_Camming.camIn(Master		  := _Front.Axis,
					   Slave		  := _Rear.Axis,
					   ActivationMode := MC_CamActivationMode.MC_CAMACTIVATION_INSTANTANEOUS,
					   Execute		  := TRUE,
					   CamTableID	  := 1);

		IF NOT _Camming.camIn.Busy AND NOT _Camming.camIn.Error THEN
			_Camming.camIn(Master := _Front.Axis, Slave := _Rear.Axis, Execute := FALSE);
			NextStep(_State);
		END_IF

	31:
		_Camming.camIn.Options.CamOperationMode := CAMOPERATIONMODE_EXCHANGE;
		_Camming.camIn.ActivationPosition		:= 250;
		_Camming.camIn(Master		  := _Front.Axis,
					   Slave		  := _Rear.Axis,
					   ActivationMode := MC_CamActivationMode.MC_CAMACTIVATION_ATMASTERAXISPOS,
					   Execute		  := TRUE,
					   CamTableID	  := 2);

		IF NOT _Camming.camIn.Busy AND NOT _Camming.camIn.Error THEN
			_Camming.camIn(Master := _Front.Axis, Slave := _Rear.Axis, Execute := FALSE);
			NextStep(_State);
		END_IF

	32:
		_Virtual.MoveRelative(_Distance);
		SetStep(_State, 30);

	51:
		_Virtual.Parameters.Velocity	 := _Speed;
		_Virtual.Parameters.Acceleration := _Acc;
		_Virtual.Parameters.Deceleration := _Dec;
		_Virtual.Parameters.Jerk		 := _Jerk;
		_Virtual.MoveRelative(1500);
		NextMinorStep(_State);

	52:
		IF NOT _Virtual.Axis.Status.CamTableQueued OR _Camming.camIn.InSync THEN
			_Camming.camIn.Options.CamOperationMode := CAMOPERATIONMODE_EXCHANGE;
			_Camming.camIn.ActivationPosition		:= 0;
			_Camming.camIn(Master		  := _Front.Axis,
						   Slave		  := _Rear.Axis,
						   ActivationMode := MC_CamActivationMode.MC_CAMACTIVATION_NEXTCYCLE,
						   Execute		  := TRUE,
						   CamTableID	  := 1);

			IF NOT _Camming.camIn.Busy AND NOT _Camming.camIn.Error THEN //If this errors/isn't instant, womp womp
				_Camming.camIn(Master := _Front.Axis, Slave := _Rear.Axis, Execute := FALSE);
				NextMinorStep(_State);
			END_IF
		END_IF

	53:
		IF NOT _Virtual.CurrentTask.Busy AND NOT _Virtual.CurrentTask.Error THEN
			NextStep(_State);
		END_IF

	60:
		_Camming.camOut(Slave := _Rear.Axis, Execute := TRUE);
		IF NOT _Camming.camOut.Busy AND NOT _Camming.camOut.Error THEN
			_Camming.camOut(Slave := _Rear.Axis, Execute := FALSE);
			SetStep(_State, 0);
		END_IF
END_CASE
END_METHOD

PROPERTY FrontMover : I_XtsMover
GET
FrontMover := _Front;
END_GET
SET
_Front := FrontMover;
END_SET
END_PROPERTY

PROPERTY RearMover : I_XtsMover
GET
RearMover := _Rear;
END_GET
SET
_Rear := RearMover;
END_SET
END_PROPERTY

METHOD Reset
_Camming.camIn(Master := _Front.Axis, Slave := _Rear.Axis, Execute := FALSE);
_Virtual.Reset();
SetStep(_State, 0);
END_METHOD

METHOD Start
NextStep(_State);
END_METHOD

{warning 'Add method implementation '}
METHOD Stop
END_METHOD

PROPERTY VirtualMover : I_XtsMover
GET
VirtualMover := _Virtual;
END_GET
SET
_Virtual := VirtualMover;
END_SET
END_PROPERTY

END_FUNCTION_BLOCK

// ---- Tests/FB_XtsBallCamBuilder.TcPOU
FUNCTION_BLOCK FB_XtsBallCamBuilder
(* Builds a TwinCAT motion-function cam table (MC_MotionFunctionPoint array) for two XTS movers that
   must keep a constant distance measured along the path of a ball mounted outward of the mover path.
   Track: straights and 180 deg modules (Beckhoff AT2050 geometry: quintic curvature ramp + circular arc).
   Layout per module: entry ramp up (POLYNOM3) - plateau (POLYNOM1) - ramp down (POLYNOM3) - line (POLYNOM1)
                      exit  ramp down (POLYNOM3) - plateau (POLYNOM1) - ramp up (POLYNOM3) - line (POLYNOM1)
   All SlaveVelo/SlaveAcc/SlaveJerk = 0 -> TwinCAT takes the ramp end velocities from the adjacent lines.
   Generated 2026-09-16 from cam_M180-1680_D115_clothoid_xlsx_min18_p3_std. *)
VAR_INPUT
	// ---- cam table range ----
	fMasterStart		: LREAL := 180.0;		// [mm] master position of the first point
	fMasterEnd			: LREAL := 1680.0;		// [mm] master position of the last point
	fBallDistance		: LREAL := 115.0;		// [mm] distance master ball -> slave ball along the ball path (slave trails the master)

	// ---- track layout in master coordinates ----
	nCurves				: UINT  := 2;			// number of 180 deg modules inside the table range
	aCurveStart			: ARRAY[1..4] OF LREAL := [250.0, 1000.0, 0.0, 0.0];	// [mm] start of each module
	fModuleLength		: LREAL := 500.0;		// [mm] module length along the mover path (AT2050: 500)
	fTransLength		: LREAL := 84.0;		// [mm] curvature transition length at each module end (quintic ramp)
	fBallOffset			: LREAL := 103.03;		// [mm] lateral offset of the ball, outward of the mover path (r_ball - r_xts)

	// ---- knot layout, offsets relative to the module start [mm] (optimised for D = 115 mm, offset 103 mm) ----
	aEntryKnots			: ARRAY[1..4] OF LREAL := [16.0, 67.5, 90.5, 134.7];	// ramp start, plateau start, plateau end, ramp end
	aExitKnots			: ARRAY[1..4] OF LREAL := [432.0, 483.0, 493.0, 603.0];	// ramp start, plateau start, plateau end, ramp end

	// ---- options ----
	bZeroEndVelocity	: BOOL  := FALSE;		// TRUE: slave at rest at the first and last point (POLYNOM5 run-up / run-down + link line)
	fLinkLength			: LREAL := 10.0;		// [mm] POLYNOM1 link between run-up/run-down and the first/last ramp

	// ---- target buffer ----
	pPoints				: POINTER TO MC_MotionFunctionPoint;	// ADR(camPoints[first element])
	nMaxPoints			: UDINT;				// number of elements in the buffer
END_VAR
VAR_OUTPUT
	nPoints				: UDINT;				// points written (use as NoOfRows)
	fArcRadius			: LREAL;				// [mm] radius of the circular middle, derived: (fModuleLength - fTransLength) / PI
	fPeakRatio			: LREAL;				// max slave/master speed ratio = 1 + fBallOffset / fArcRadius
	bError				: BOOL;
	sError				: STRING(255);
END_VAR
VAR
	fKMax				: LREAL;				// [1/mm] curvature of the circular middle
END_VAR
VAR CONSTANT
	fPI					: LREAL := 3.14159265358979;
END_VAR

(* nothing cyclic: call Build() once *)

METHOD PRIVATE AddPoint
VAR_INPUT
	fMaster	: LREAL;
	eFunc	: MC_MotionFunctionType;
END_VAR
IF bError THEN RETURN; END_IF
IF nPoints >= nMaxPoints THEN
	bError := TRUE; sError := 'point buffer too small'; RETURN;
END_IF
IF nPoints > 0 AND_THEN fMaster <= pPoints[nPoints - 1].MasterPos THEN
	bError := TRUE; sError := CONCAT('master positions not increasing at point ', UDINT_TO_STRING(nPoints + 1)); RETURN;
END_IF

pPoints[nPoints].PointIndex        := nPoints + 1;
pPoints[nPoints].MasterPos         := fMaster;
pPoints[nPoints].SlavePos          := SlavePos(fMaster);
pPoints[nPoints].FunctionType      := eFunc;
pPoints[nPoints].PointType         := SEL(nPoints = 0, MC_MotionPointType.MOTIONPOINTTYPE_MOTION, MC_MotionPointType.MOTIONPOINTTYPE_ACTIVATION);
pPoints[nPoints].RelIndexNextPoint := 1;
pPoints[nPoints].SlaveVelo         := 0.0;
pPoints[nPoints].SlaveAcc          := 0.0;
pPoints[nPoints].SlaveJerk         := 0.0;
nPoints := nPoints + 1;
END_METHOD

METHOD PRIVATE BallArc : LREAL
(* path length of the ball for mover position fS: B(s) = s + d * theta(s) *)
VAR_INPUT
	fS	: LREAL;
END_VAR
BallArc := fS + fBallOffset * Theta(fS);
END_METHOD

METHOD Build : BOOL
VAR
	nCurve	: UINT;
	fC		: LREAL;
END_VAR
bError := FALSE; sError := ''; nPoints := 0;

IF pPoints = 0 OR nMaxPoints < 2 THEN
	bError := TRUE; sError := 'pPoints / nMaxPoints not set'; RETURN;
END_IF
IF nCurves < 1 OR nCurves > 4 THEN
	bError := TRUE; sError := 'nCurves must be 1..4'; RETURN;
END_IF
IF fTransLength <= 0 OR fTransLength >= 0.5 * fModuleLength THEN
	bError := TRUE; sError := 'fTransLength out of range'; RETURN;
END_IF

// 180 deg over the module: kmax * (L_mod - L_trans) = PI  (the quintic ramp integrates to half its length)
fKMax      := fPI / (fModuleLength - fTransLength);
fArcRadius := 1.0 / fKMax;
fPeakRatio := 1.0 + fBallOffset * fKMax;

// ---- first point(s) ----
IF bZeroEndVelocity THEN
	AddPoint(fMasterStart, MC_MotionFunctionType.MOTIONFUNCTYPE_POLYNOM5);								// run-up from rest
	AddPoint(aCurveStart[1] + aEntryKnots[1] - fLinkLength, MC_MotionFunctionType.MOTIONFUNCTYPE_POLYNOM1);	// short line
ELSE
	AddPoint(fMasterStart, MC_MotionFunctionType.MOTIONFUNCTYPE_POLYNOM1);
END_IF

// ---- per module: entry (ratio 1 -> peak -> 1) and exit (ratio 1 -> 1/peak -> 1) ----
FOR nCurve := 1 TO nCurves DO
	fC := aCurveStart[nCurve];
	AddPoint(fC + aEntryKnots[1], MC_MotionFunctionType.MOTIONFUNCTYPE_POLYNOM3);	// ramp up
	AddPoint(fC + aEntryKnots[2], MC_MotionFunctionType.MOTIONFUNCTYPE_POLYNOM1);	// plateau at the ratio maximum
	AddPoint(fC + aEntryKnots[3], MC_MotionFunctionType.MOTIONFUNCTYPE_POLYNOM3);	// ramp down
	AddPoint(fC + aEntryKnots[4], MC_MotionFunctionType.MOTIONFUNCTYPE_POLYNOM1);	// both on the arc: ratio 1
	AddPoint(fC + aExitKnots[1],  MC_MotionFunctionType.MOTIONFUNCTYPE_POLYNOM3);	// ramp down
	AddPoint(fC + aExitKnots[2],  MC_MotionFunctionType.MOTIONFUNCTYPE_POLYNOM1);	// plateau at the ratio minimum
	AddPoint(fC + aExitKnots[3],  MC_MotionFunctionType.MOTIONFUNCTYPE_POLYNOM3);	// ramp up
	AddPoint(fC + aExitKnots[4],  MC_MotionFunctionType.MOTIONFUNCTYPE_POLYNOM1);	// both on the straight: ratio 1
END_FOR

// ---- last point(s) ----
IF bZeroEndVelocity THEN
	AddPoint(aCurveStart[nCurves] + aExitKnots[4] + fLinkLength, MC_MotionFunctionType.MOTIONFUNCTYPE_POLYNOM5);	// run-down to rest
END_IF
AddPoint(fMasterEnd, MC_MotionFunctionType.MOTIONFUNCTYPE_POLYNOM1);

IF NOT bError THEN
	pPoints[nPoints - 1].RelIndexNextPoint := 0;	// terminate the table
END_IF
Build := NOT bError;
END_METHOD

METHOD PRIVATE InvBallArc : LREAL
(* mover position for a ball path length: Newton iteration on B(s) = fB *)
VAR_INPUT
	fB	: LREAL;
END_VAR
VAR
	fS, fF	: LREAL;
	i		: UINT;
END_VAR
fS := fB;
FOR i := 1 TO 50 DO
	fF := BallArc(fS) - fB;
	IF ABS(fF) < 1.0E-9 THEN EXIT; END_IF
	fS := fS - fF / (1.0 + fBallOffset * Kappa(fS));
END_FOR
InvBallArc := fS;
END_METHOD

METHOD PRIVATE Kappa : LREAL
(* curvature [1/mm] of the mover path at fS *)
VAR_INPUT
	fS	: LREAL;
END_VAR
VAR
	i	: UINT;
END_VAR
Kappa := 0.0;
FOR i := 1 TO nCurves DO
	Kappa := Kappa + KappaMod(fS - aCurveStart[i]);
END_FOR
END_METHOD

METHOD PRIVATE KappaMod : LREAL
(* curvature inside one 180 deg module, fU = position from module start.
   Quintic ramp k = kmax * (10 t^3 - 15 t^4 + 6 t^5), t = u / L_trans; circular middle; mirrored ramp *)
VAR_INPUT
	fU	: LREAL;
END_VAR
VAR
	t	: LREAL;
END_VAR
IF fU <= 0.0 OR fU >= fModuleLength THEN
	KappaMod := 0.0;
ELSIF fU < fTransLength THEN
	t := fU / fTransLength;
	KappaMod := fKMax * t * t * t * (10.0 - 15.0 * t + 6.0 * t * t);
ELSIF fU <= fModuleLength - fTransLength THEN
	KappaMod := fKMax;
ELSE
	t := (fModuleLength - fU) / fTransLength;
	KappaMod := fKMax * t * t * t * (10.0 - 15.0 * t + 6.0 * t * t);
END_IF
END_METHOD

METHOD SlavePos : LREAL
(* exact slave position for a master position: constant distance fBallDistance along the ball path *)
VAR_INPUT
	fMaster	: LREAL;
END_VAR
SlavePos := InvBallArc(BallArc(fMaster) - fBallDistance);
END_METHOD

METHOD SpeedRatio : LREAL
(* exact slave/master speed ratio ds/dm for a master position (diagnostics) *)
VAR_INPUT
	fMaster	: LREAL;
END_VAR
SpeedRatio := (1.0 + fBallOffset * Kappa(fMaster)) / (1.0 + fBallOffset * Kappa(SlavePos(fMaster)));
END_METHOD

METHOD PRIVATE Theta : LREAL
(* heading angle [rad] turned between fMasterStart and fS (sum over the modules; table covers one lap) *)
VAR_INPUT
	fS	: LREAL;
END_VAR
VAR
	i	: UINT;
END_VAR
Theta := 0.0;
FOR i := 1 TO nCurves DO
	Theta := Theta + ThetaMod(fS - aCurveStart[i]);
END_FOR
END_METHOD

METHOD PRIVATE ThetaMod : LREAL
(* heading [rad] turned inside one module up to fU (closed-form integral of KappaMod):
   ramp: kmax * L_trans * (2.5 t^4 - 3 t^5 + t^6); a full ramp turns kmax * L_trans / 2 *)
VAR_INPUT
	fU	: LREAL;
END_VAR
VAR
	t	: LREAL;
END_VAR
IF fU <= 0.0 THEN
	ThetaMod := 0.0;
ELSIF fU >= fModuleLength THEN
	ThetaMod := fPI;
ELSIF fU < fTransLength THEN
	t := fU / fTransLength;
	ThetaMod := fKMax * fTransLength * t * t * t * t * (2.5 - 3.0 * t + t * t);
ELSIF fU <= fModuleLength - fTransLength THEN
	ThetaMod := 0.5 * fKMax * fTransLength + fKMax * (fU - fTransLength);
ELSE
	t := (fModuleLength - fU) / fTransLength;
	ThetaMod := fPI - fKMax * fTransLength * t * t * t * t * (2.5 - 3.0 * t + t * t);
END_IF
END_METHOD

END_FUNCTION_BLOCK
